// TIA Portal project "Green_Finished" (V17)
// Vorlageprojekt für das Buch mit Zielsystem S7-1200

(* hardware
DEVICE "S7-1200-Station_1"  S7-1200 Station
   slot 0: "Baugruppenträger_0"  Rack  V1.0
   slot 1: "PLC_1"  CPU 1211C DC/DC/DC  6ES7 211-1AE40-0XB0  V4.1
*)

// ===== PLC "PLC_1"  CPU 1211C DC/DC/DC =====

VAR_GLOBAL   // PLC tag table "Standard-Variablentabelle"
   "Tag_1" AT %M0.0 : Bool;
   "Tag_2" AT %M0.1 : Bool;
   "Tag_3" AT %M0.2 : Bool;
   "Tag_4" AT %M0.3 : Bool;
   "Tag_5" AT %M0.4 : Bool;
   "Tag_6" AT %M0.5 : Bool;
   "Tag_7" AT %M0.6 : Bool;
   "vision 0" AT %I2.2 : Bool;
   "arm 0 turn" AT %Q1.5 : Bool;
   "arm 0 +" AT %Q1.6 : Bool;
   "arm 1 turn" AT %Q1.7 : Bool;
   "arm 1 +" AT %Q2.0 : Bool;
   "arm 2 turn" AT %Q2.1 : Bool;
   "arm 2 +" AT %Q2.2 : Bool;
   "6m belt 1" AT %Q2.3 : Bool;
   "curved belt 1" AT %Q2.4 : Bool;
   "4m belt 2" AT %Q2.6 : Bool;
   "vision difuse" AT %I2.3 : Bool;
   "machine 0 produce lid" AT %Q3.1 : Bool;
   "machine 0 start" AT %Q3.2 : Bool;
   "macine 0 stop" AT %Q3.3 : Bool;
   "machine busy" AT %I1.7 : Bool;
   "machine 1 start" AT %Q3.5 : Bool;
   "machine 1 stop" AT %Q3.6 : Bool;
   "machine 1 produce lid" AT %Q3.4 : Bool;
   "curved belt 3" AT %Q4.2 : Bool;
   "curved belt 2" AT %Q4.1 : Bool;
   "6m belt 3" AT %Q4.0 : Bool;
   "6m belt 2" AT %Q3.7 : Bool;
   "4m belt 3" AT %Q3.0 : Bool;
   "2m belt 1" AT %Q2.7 : Bool;
   "2m belt 0" AT %Q2.5 : Bool;
   "diffuse belt 1" AT %I1.6 : Bool;
   "diffuse belt 1 second" AT %I2.5 : Bool;
   "diffuse belt 2" AT %I2.1 : Bool;
   "diffuse belt 2 second" AT %I2.4 : Bool;
   "machine 2 produce lid" AT %Q4.3 : Bool;
   "machine 2 start" AT %Q4.4 : Bool;
   "machine 2 stop" AT %Q4.5 : Bool;
   "machine 3 produce lid" AT %Q4.6 : Bool;
   "machine 3 start" AT %Q4.7 : Bool;
   "machine 3 stop" AT %Q5.0 : Bool;
   "Tag_8" AT %M3.2 : Bool;
   "Tag_9" AT %M3.3 : Bool;
   "Tag_10" AT %M8.0 : Bool;
   "Tag_11" AT %M3.4 : Bool;
   "Tag_12" AT %M3.5 : Bool;
   "Tag_13" AT %M3.6 : Bool;
   "Tag_14" AT %M3.7 : Bool;
   "Tag_15" AT %M4.0 : Bool;
END_VAR

VAR_GLOBAL   // PLC tag table "Sensors & Pushbuttons"
   "Start" AT %I0.0 : Bool;
   "Stop" AT %I0.1 : Bool;
   "Emergency Stop" AT %I0.2 : Bool;
   "RobotDetect" AT %I0.3 : Bool;
   "Diffuser 1" AT %I0.4 : Bool;
   "Diffuser 2" AT %I0.5 : Bool;
   "Frontlimit0" AT %I0.6 : Bool;
   "Backlimit0" AT %I0.7 : Bool;
   "Frontlimit1" AT %I1.0 : Bool;
   "Backlimit1" AT %I1.1 : Bool;
   "Diffuser 3" AT %I1.2 : Bool;
   "Zmoving" AT %I1.3 : Bool;
   "Xmoving" AT %I1.4 : Bool;
   "OBJheld" AT %I1.5 : Bool;
   "Diffuser 9" AT %I3.0 : Bool;
   "Diffuser 10" AT %I3.1 : Bool;
   "Diffuser 13" AT %I3.2 : Bool;
   "Diffuser 14" AT %I3.3 : Bool;
   "Robot1zmoving" AT %I3.4 : Bool;
   "Robot1Xmoving" AT %I3.5 : Bool;
   "ClamperLimit" AT %I4.0 : Bool;
   "ClamperClamped" AT %I4.1 : Bool;
   "Robot1Detected" AT %I3.6 : Bool;
   "Diffuser 17" AT %I4.2 : Bool;
   "Diiffuser 18" AT %I4.3 : Bool;
END_VAR

VAR_GLOBAL   // PLC tag table "Actuators"
   "FeedingConveyer" AT %Q0.0 : Bool;
   "Bridge" AT %Q0.1 : Bool;
   "To machine" AT %Q0.2 : Bool;
   "CurvedConveyer" AT %Q0.3 : Bool;
   "Emitter" AT %Q0.4 : Bool;
   "Pusher0" AT %Q0.5 : Bool;
   "Pusher1" AT %Q0.6 : Bool;
   "GreenLight" AT %Q0.7 : Bool;
   "RedLight" AT %Q1.0 : Bool;
   "Xcontrol" AT %Q1.1 : Bool;
   "Zcontrol" AT %Q1.2 : Bool;
   "Grab" AT %Q1.3 : Bool;
   "WarningLight" AT %Q1.4 : Bool;
   "Belt4m4" AT %Q5.5 : Bool;
   "Belt4m8" AT %Q5.6 : Bool;
   "Cbc4cw" AT %Q5.7 : Bool;
   "Belt6m4" AT %Q6.0 : Bool;
   "Belt4m5" AT %Q6.2 : Bool;
   "CBC5cw" AT %Q6.3 : Bool;
   "Belt2m2" AT %Q6.4 : Bool;
   "cbc5ccw" AT %Q6.5 : Bool;
   "belt6m5" AT %Q6.6 : Bool;
   "Robot1z" AT %Q7.0 : Bool;
   "Robot1x" AT %Q7.5 : Bool;
   "Robot1grab" AT %Q7.3 : Bool;
   "ClamperRaise" AT %Q8.1 : Bool;
   "ClamperClamp" AT %Q8.0 : Bool;
END_VAR

FUNCTION "MHJ-PLC-Lab-Function-S71200" : Void   // FC9000, SCL
{ S7_Optimized_Access := 'TRUE' }
VERSION : 0.1
   VAR_TEMP
      rdTimeReturn : Int;
      outputTime : DTL;
      SyncVal : Byte;
      forVal : Int;
      forVal_2 : Int;
      Value : Byte;
   END_VAR
   VAR CONSTANT
      CompVal : Byte := 16#34;
      Value_01 : Byte := 16#11;
      Value_01_DW : DWord := 16#A165_D992;
      Value_02_DW : DWord := 16#58BE_4401;
   END_VAR
BEGIN

   #Value:=PEEK(area := 16#82,
        dbNumber := 0,
        byteOffset := 511);
   #Value := #Value + 1;

   POKE(area := 16#82,
        dbNumber := 0,
        byteOffset := 511,
        value := #Value);

   POKE(area:=16#81,
        dbNumber:=0,
        byteOffset:=1016,
        value:=#Value_01_DW);
   POKE(area := 16#81,
        dbNumber := 0,
        byteOffset := 1020,
        value := #Value_02_DW);

   POKE(area := 16#81,
        dbNumber := 0,
        byteOffset := 511,
        value := B#16#00);

   FOR #forVal := 0 TO 120 DO
       FOR #forVal_2:=0 TO 10 DO
           #rdTimeReturn:=RD_SYS_T(#outputTime);
           #rdTimeReturn := WR_SYS_T(#outputTime);
           #rdTimeReturn := RD_SYS_T(#outputTime);
           #rdTimeReturn := WR_SYS_T(#outputTime);
       END_FOR;
       #SyncVal:= PEEK(area := 16#81,
                      dbNumber := 0,
                      byteOffset := 511);
       IF #SyncVal = #CompVal THEN
          GOTO M_1;
       END_IF;
   END_FOR;
   RETURN;

   M_1:
   POKE(area := 16#81,
        dbNumber := 0,
        byteOffset := 511,
        value := B#16#0);
END_FUNCTION

ORGANIZATION_BLOCK "Main"   // OB1, LAD, ProgramCycle
TITLE = "Main Program Sweep (Cycle)"
{ S7_Optimized_Access := 'TRUE' }
VERSION : 0.1
   VAR_INPUT
      Initial_Call : Bool;   // Initial call of this OB
      Remanence : Bool;   // =True, if remanent data are available
   END_VAR
   VAR_TEMP   // added for the SCL form of the ladder/FBD networks
      _w1 : Bool;
      _w2 : Bool;
      _w3 : Bool;
      _w4 : Bool;
      _w5 : Bool;
   END_VAR
BEGIN

REGION Network 1: Konnektierungsbaustein für PLC-Lab
   // Im Netzwerk 1 wird der Konnektierungsbaustein für PLC-Lab aufgerufen.
   // Dieser Aufruf darf nicht entfernt werden!
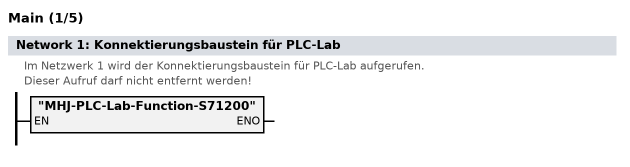
   RUNG wire#powerrail
      "MHJ-PLC-Lab-Function-S71200"()
   END_RUNG
   // the same network as SCL:
   "MHJ-PLC-Lab-Function-S71200"();
END_REGION

REGION Network 2: Ihr Programm / Conveyer Control
   // Schreiben Sie ab Netzwerk 2 Ihr Programm
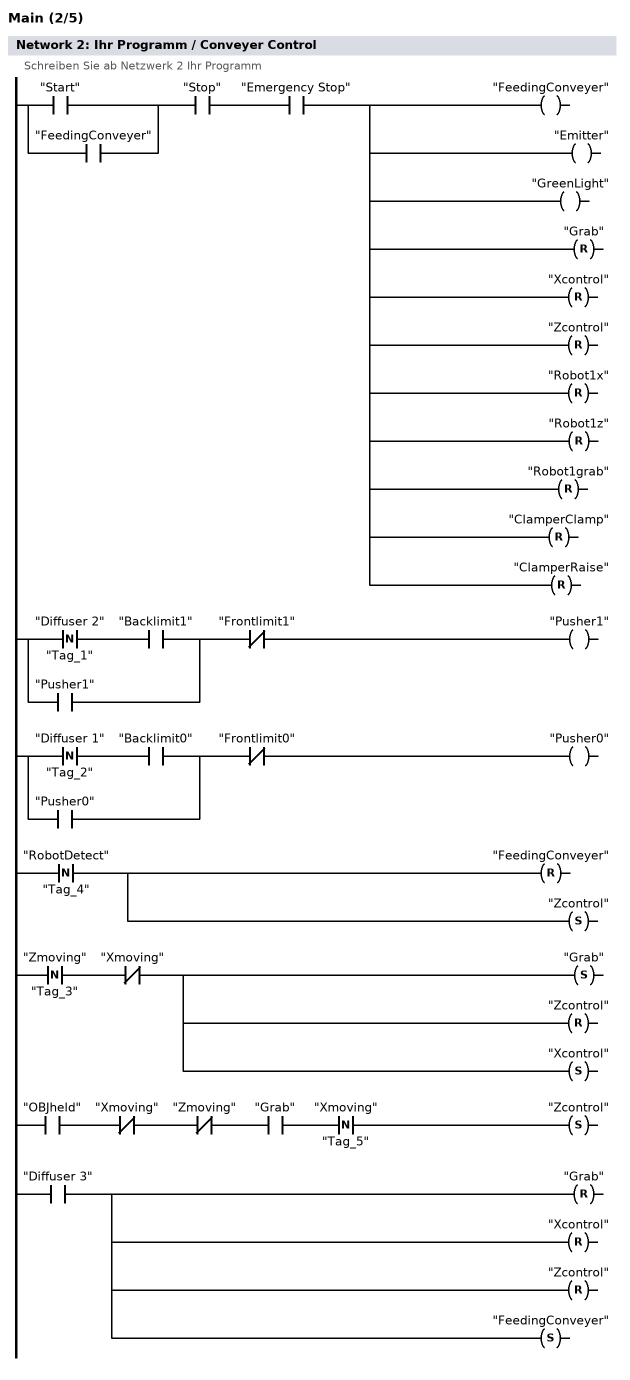
   RUNG wire#powerrail
      Contact( "Start" )
      wire#w1
      Contact( "Stop" )
      Contact( "Emergency Stop" )
      wire#w2
      Coil( "FeedingConveyer" )
   END_RUNG
   RUNG wire#powerrail
      Contact( "FeedingConveyer" )
   END_RUNG wire#w1
   RUNG wire#w2
      Coil( "Emitter" )
   END_RUNG
   RUNG wire#w2
      Coil( "GreenLight" )
   END_RUNG
   RUNG wire#w2
      R_Coil( "Grab" )
   END_RUNG
   RUNG wire#w2
      R_Coil( "Xcontrol" )
   END_RUNG
   RUNG wire#w2
      R_Coil( "Zcontrol" )
   END_RUNG
   RUNG wire#w2
      R_Coil( "Robot1x" )
   END_RUNG
   RUNG wire#w2
      R_Coil( "Robot1z" )
   END_RUNG
   RUNG wire#w2
      R_Coil( "Robot1grab" )
   END_RUNG
   RUNG wire#w2
      R_Coil( "ClamperClamp" )
   END_RUNG
   RUNG wire#w2
      R_Coil( "ClamperRaise" )
   END_RUNG
   RUNG wire#powerrail
      N_Contact(operand := "Diffuser 2", bit := "Tag_1")
      Contact( "Backlimit1" )
      wire#w3
      I_Contact( "Frontlimit1" )
      Coil( "Pusher1" )
   END_RUNG
   RUNG wire#powerrail
      Contact( "Pusher1" )
   END_RUNG wire#w3
   RUNG wire#powerrail
      N_Contact(operand := "Diffuser 1", bit := "Tag_2")
      Contact( "Backlimit0" )
      wire#w4
      I_Contact( "Frontlimit0" )
      Coil( "Pusher0" )
   END_RUNG
   RUNG wire#powerrail
      Contact( "Pusher0" )
   END_RUNG wire#w4
   RUNG wire#powerrail
      N_Contact(operand := "RobotDetect", bit := "Tag_4")
      wire#w5
      R_Coil( "FeedingConveyer" )
   END_RUNG
   RUNG wire#w5
      S_Coil( "Zcontrol" )
   END_RUNG
   RUNG wire#powerrail
      N_Contact(operand := "Zmoving", bit := "Tag_3")
      I_Contact( "Xmoving" )
      wire#w6
      S_Coil( "Grab" )
   END_RUNG
   RUNG wire#w6
      R_Coil( "Zcontrol" )
   END_RUNG
   RUNG wire#w6
      S_Coil( "Xcontrol" )
   END_RUNG
   RUNG wire#powerrail
      Contact( "OBJheld" )
      I_Contact( "Xmoving" )
      I_Contact( "Zmoving" )
      Contact( "Grab" )
      N_Contact(operand := "Xmoving", bit := "Tag_5")
      S_Coil( "Zcontrol" )
   END_RUNG
   RUNG wire#powerrail
      Contact( "Diffuser 3" )
      wire#w7
      R_Coil( "Grab" )
   END_RUNG
   RUNG wire#w7
      R_Coil( "Xcontrol" )
   END_RUNG
   RUNG wire#w7
      R_Coil( "Zcontrol" )
   END_RUNG
   RUNG wire#w7
      S_Coil( "FeedingConveyer" )
   END_RUNG
   // the same network as SCL:
   "FeedingConveyer" := ("Start" OR "FeedingConveyer") AND "Stop" AND "Emergency Stop";
   "Emitter" := "FeedingConveyer";
   "GreenLight" := "FeedingConveyer";
   IF "FeedingConveyer" THEN
       "Grab" := FALSE;
       "Xcontrol" := FALSE;
       "Zcontrol" := FALSE;
       "Robot1x" := FALSE;
       "Robot1z" := FALSE;
       "Robot1grab" := FALSE;
       "ClamperClamp" := FALSE;
       "ClamperRaise" := FALSE;
   END_IF;
   #_w1 := NOT "Diffuser 2" AND "Tag_1";   // falling edge of "Diffuser 2"
   "Tag_1" := "Diffuser 2";
   "Pusher1" := ((#_w1 AND "Backlimit1") OR "Pusher1") AND NOT "Frontlimit1";
   #_w2 := NOT "Diffuser 1" AND "Tag_2";   // falling edge of "Diffuser 1"
   "Tag_2" := "Diffuser 1";
   "Pusher0" := ((#_w2 AND "Backlimit0") OR "Pusher0") AND NOT "Frontlimit0";
   #_w3 := NOT "RobotDetect" AND "Tag_4";   // falling edge of "RobotDetect"
   "Tag_4" := "RobotDetect";
   IF #_w3 THEN
       "FeedingConveyer" := FALSE;
       "Zcontrol" := TRUE;
   END_IF;
   #_w4 := NOT "Zmoving" AND "Tag_3";   // falling edge of "Zmoving"
   "Tag_3" := "Zmoving";
   IF #_w4 AND NOT "Xmoving" THEN
       "Grab" := TRUE;
       "Zcontrol" := FALSE;
       "Xcontrol" := TRUE;
   END_IF;
   #_w5 := "OBJheld" AND NOT "Xmoving" AND NOT "Zmoving" AND "Grab" AND NOT "Xmoving" AND "Tag_5";   // falling edge of "Xmoving"
   "Tag_5" := "Xmoving";
   IF #_w5 THEN "Zcontrol" := TRUE; END_IF;
   IF "Diffuser 3" THEN
       "Grab" := FALSE;
       "Xcontrol" := FALSE;
       "Zcontrol" := FALSE;
       "FeedingConveyer" := TRUE;
   END_IF;
END_REGION

REGION Network 3
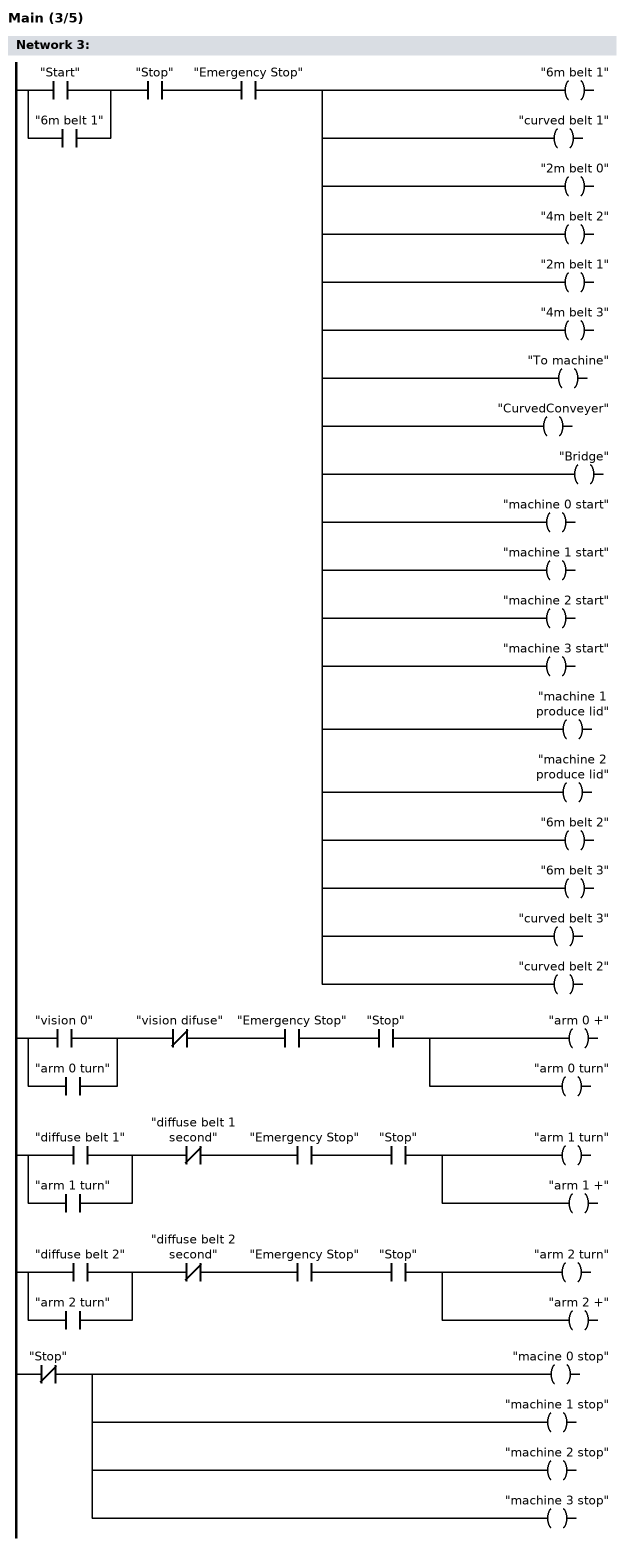
   RUNG wire#powerrail
      Contact( "Start" )
      wire#w1
      Contact( "Stop" )
      Contact( "Emergency Stop" )
      wire#w2
      Coil( "6m belt 1" )
   END_RUNG
   RUNG wire#powerrail
      Contact( "6m belt 1" )
   END_RUNG wire#w1
   RUNG wire#w2
      Coil( "curved belt 1" )
   END_RUNG
   RUNG wire#w2
      Coil( "2m belt 0" )
   END_RUNG
   RUNG wire#w2
      Coil( "4m belt 2" )
   END_RUNG
   RUNG wire#w2
      Coil( "2m belt 1" )
   END_RUNG
   RUNG wire#w2
      Coil( "4m belt 3" )
   END_RUNG
   RUNG wire#w2
      Coil( "To machine" )
   END_RUNG
   RUNG wire#w2
      Coil( "CurvedConveyer" )
   END_RUNG
   RUNG wire#w2
      Coil( "Bridge" )
   END_RUNG
   RUNG wire#w2
      Coil( "machine 0 start" )
   END_RUNG
   RUNG wire#w2
      Coil( "machine 1 start" )
   END_RUNG
   RUNG wire#w2
      Coil( "machine 2 start" )
   END_RUNG
   RUNG wire#w2
      Coil( "machine 3 start" )
   END_RUNG
   RUNG wire#w2
      Coil( "machine 1 produce lid" )
   END_RUNG
   RUNG wire#w2
      Coil( "machine 2 produce lid" )
   END_RUNG
   RUNG wire#w2
      Coil( "6m belt 2" )
   END_RUNG
   RUNG wire#w2
      Coil( "6m belt 3" )
   END_RUNG
   RUNG wire#w2
      Coil( "curved belt 3" )
   END_RUNG
   RUNG wire#w2
      Coil( "curved belt 2" )
   END_RUNG
   RUNG wire#powerrail
      Contact( "vision 0" )
      wire#w3
      I_Contact( "vision difuse" )
      Contact( "Emergency Stop" )
      Contact( "Stop" )
      wire#w4
      Coil( "arm 0 +" )
   END_RUNG
   RUNG wire#powerrail
      Contact( "arm 0 turn" )
   END_RUNG wire#w3
   RUNG wire#w4
      Coil( "arm 0 turn" )
   END_RUNG
   RUNG wire#powerrail
      Contact( "diffuse belt 1" )
      wire#w5
      I_Contact( "diffuse belt 1 second" )
      Contact( "Emergency Stop" )
      Contact( "Stop" )
      wire#w6
      Coil( "arm 1 turn" )
   END_RUNG
   RUNG wire#powerrail
      Contact( "arm 1 turn" )
   END_RUNG wire#w5
   RUNG wire#w6
      Coil( "arm 1 +" )
   END_RUNG
   RUNG wire#powerrail
      Contact( "diffuse belt 2" )
      wire#w7
      I_Contact( "diffuse belt 2 second" )
      Contact( "Emergency Stop" )
      Contact( "Stop" )
      wire#w8
      Coil( "arm 2 turn" )
   END_RUNG
   RUNG wire#powerrail
      Contact( "arm 2 turn" )
   END_RUNG wire#w7
   RUNG wire#w8
      Coil( "arm 2 +" )
   END_RUNG
   RUNG wire#powerrail
      I_Contact( "Stop" )
      wire#w9
      Coil( "macine 0 stop" )
   END_RUNG
   RUNG wire#w9
      Coil( "machine 1 stop" )
   END_RUNG
   RUNG wire#w9
      Coil( "machine 2 stop" )
   END_RUNG
   RUNG wire#w9
      Coil( "machine 3 stop" )
   END_RUNG
   // the same network as SCL:
   "6m belt 1" := ("Start" OR "6m belt 1") AND "Stop" AND "Emergency Stop";
   "curved belt 1" := "6m belt 1";
   "2m belt 0" := "6m belt 1";
   "4m belt 2" := "6m belt 1";
   "2m belt 1" := "6m belt 1";
   "4m belt 3" := "6m belt 1";
   "To machine" := "6m belt 1";
   "CurvedConveyer" := "6m belt 1";
   "Bridge" := "6m belt 1";
   "machine 0 start" := "6m belt 1";
   "machine 1 start" := "6m belt 1";
   "machine 2 start" := "6m belt 1";
   "machine 3 start" := "6m belt 1";
   "machine 1 produce lid" := "6m belt 1";
   "machine 2 produce lid" := "6m belt 1";
   "6m belt 2" := "6m belt 1";
   "6m belt 3" := "6m belt 1";
   "curved belt 3" := "6m belt 1";
   "curved belt 2" := "6m belt 1";
   "arm 0 +" := ("vision 0" OR "arm 0 turn") AND NOT "vision difuse" AND "Emergency Stop" AND "Stop";
   "arm 0 turn" := "arm 0 +";
   "arm 1 turn" := ("diffuse belt 1" OR "arm 1 turn") AND NOT "diffuse belt 1 second" AND "Emergency Stop" AND "Stop";
   "arm 1 +" := "arm 1 turn";
   "arm 2 turn" := ("diffuse belt 2" OR "arm 2 turn") AND NOT "diffuse belt 2 second" AND "Emergency Stop" AND "Stop";
   "arm 2 +" := "arm 2 turn";
   "macine 0 stop" := NOT "Stop";
   "machine 1 stop" := NOT "Stop";
   "machine 2 stop" := NOT "Stop";
   "machine 3 stop" := NOT "Stop";
END_REGION

REGION Network 4
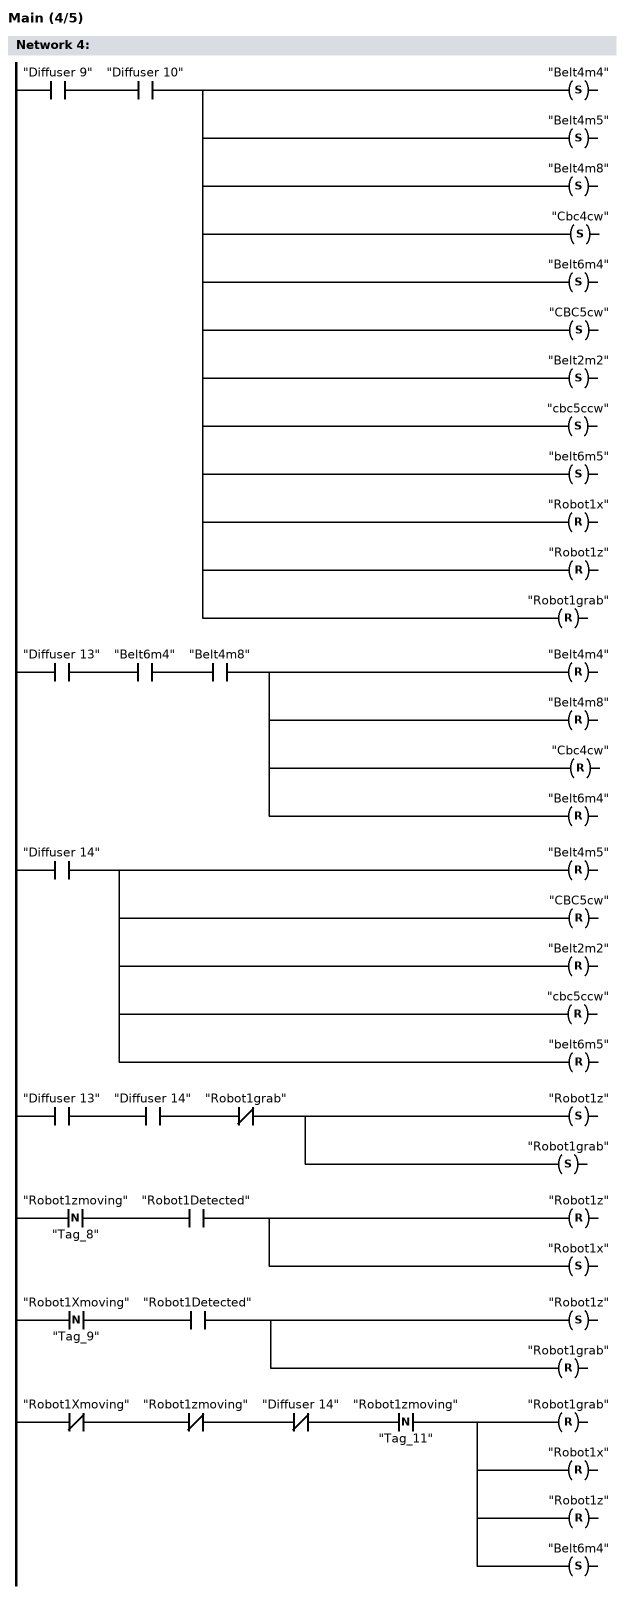
   RUNG wire#powerrail
      Contact( "Diffuser 9" )
      Contact( "Diffuser 10" )
      wire#w1
      S_Coil( "Belt4m4" )
   END_RUNG
   RUNG wire#w1
      S_Coil( "Belt4m5" )
   END_RUNG
   RUNG wire#w1
      S_Coil( "Belt4m8" )
   END_RUNG
   RUNG wire#w1
      S_Coil( "Cbc4cw" )
   END_RUNG
   RUNG wire#w1
      S_Coil( "Belt6m4" )
   END_RUNG
   RUNG wire#w1
      S_Coil( "CBC5cw" )
   END_RUNG
   RUNG wire#w1
      S_Coil( "Belt2m2" )
   END_RUNG
   RUNG wire#w1
      S_Coil( "cbc5ccw" )
   END_RUNG
   RUNG wire#w1
      S_Coil( "belt6m5" )
   END_RUNG
   RUNG wire#w1
      R_Coil( "Robot1x" )
   END_RUNG
   RUNG wire#w1
      R_Coil( "Robot1z" )
   END_RUNG
   RUNG wire#w1
      R_Coil( "Robot1grab" )
   END_RUNG
   RUNG wire#powerrail
      Contact( "Diffuser 13" )
      Contact( "Belt6m4" )
      Contact( "Belt4m8" )
      wire#w2
      R_Coil( "Belt4m4" )
   END_RUNG
   RUNG wire#w2
      R_Coil( "Belt4m8" )
   END_RUNG
   RUNG wire#w2
      R_Coil( "Cbc4cw" )
   END_RUNG
   RUNG wire#w2
      R_Coil( "Belt6m4" )
   END_RUNG
   RUNG wire#powerrail
      Contact( "Diffuser 14" )
      wire#w3
      R_Coil( "Belt4m5" )
   END_RUNG
   RUNG wire#w3
      R_Coil( "CBC5cw" )
   END_RUNG
   RUNG wire#w3
      R_Coil( "Belt2m2" )
   END_RUNG
   RUNG wire#w3
      R_Coil( "cbc5ccw" )
   END_RUNG
   RUNG wire#w3
      R_Coil( "belt6m5" )
   END_RUNG
   RUNG wire#powerrail
      Contact( "Diffuser 13" )
      Contact( "Diffuser 14" )
      I_Contact( "Robot1grab" )
      wire#w4
      S_Coil( "Robot1z" )
   END_RUNG
   RUNG wire#w4
      S_Coil( "Robot1grab" )
   END_RUNG
   RUNG wire#powerrail
      N_Contact(operand := "Robot1zmoving", bit := "Tag_8")
      Contact( "Robot1Detected" )
      wire#w5
      R_Coil( "Robot1z" )
   END_RUNG
   RUNG wire#w5
      S_Coil( "Robot1x" )
   END_RUNG
   RUNG wire#powerrail
      N_Contact(operand := "Robot1Xmoving", bit := "Tag_9")
      Contact( "Robot1Detected" )
      wire#w6
      S_Coil( "Robot1z" )
   END_RUNG
   RUNG wire#w6
      R_Coil( "Robot1grab" )
   END_RUNG
   RUNG wire#powerrail
      I_Contact( "Robot1Xmoving" )
      I_Contact( "Robot1zmoving" )
      I_Contact( "Diffuser 14" )
      N_Contact(operand := "Robot1zmoving", bit := "Tag_11")
      wire#w7
      R_Coil( "Robot1grab" )
   END_RUNG
   RUNG wire#w7
      R_Coil( "Robot1x" )
   END_RUNG
   RUNG wire#w7
      R_Coil( "Robot1z" )
   END_RUNG
   RUNG wire#w7
      S_Coil( "Belt6m4" )
   END_RUNG
   // the same network as SCL:
   IF "Diffuser 9" AND "Diffuser 10" THEN
       "Belt4m4" := TRUE;
       "Belt4m5" := TRUE;
       "Belt4m8" := TRUE;
       "Cbc4cw" := TRUE;
       "Belt6m4" := TRUE;
       "CBC5cw" := TRUE;
       "Belt2m2" := TRUE;
       "cbc5ccw" := TRUE;
       "belt6m5" := TRUE;
       "Robot1x" := FALSE;
       "Robot1z" := FALSE;
       "Robot1grab" := FALSE;
   END_IF;
   IF "Diffuser 13" AND "Belt6m4" AND "Belt4m8" THEN "Belt4m4" := FALSE; END_IF;
   #_w1 := "Diffuser 13" AND "Belt6m4" AND "Belt4m8";
   IF #_w1 THEN
       "Belt4m8" := FALSE;
       "Cbc4cw" := FALSE;
       "Belt6m4" := FALSE;
   END_IF;
   IF "Diffuser 14" THEN
       "Belt4m5" := FALSE;
       "CBC5cw" := FALSE;
       "Belt2m2" := FALSE;
       "cbc5ccw" := FALSE;
       "belt6m5" := FALSE;
   END_IF;
   IF "Diffuser 13" AND "Diffuser 14" AND NOT "Robot1grab" THEN
       "Robot1z" := TRUE;
       "Robot1grab" := TRUE;
   END_IF;
   #_w2 := NOT "Robot1zmoving" AND "Tag_8";   // falling edge of "Robot1zmoving"
   "Tag_8" := "Robot1zmoving";
   IF #_w2 AND "Robot1Detected" THEN
       "Robot1z" := FALSE;
       "Robot1x" := TRUE;
   END_IF;
   #_w3 := NOT "Robot1Xmoving" AND "Tag_9";   // falling edge of "Robot1Xmoving"
   "Tag_9" := "Robot1Xmoving";
   IF #_w3 AND "Robot1Detected" THEN
       "Robot1z" := TRUE;
       "Robot1grab" := FALSE;
   END_IF;
   #_w4 := NOT "Robot1Xmoving" AND NOT "Robot1zmoving" AND NOT "Diffuser 14" AND NOT "Robot1zmoving" AND "Tag_11";   // falling edge of "Robot1zmoving"
   "Tag_11" := "Robot1zmoving";
   IF #_w4 THEN
       "Robot1grab" := FALSE;
       "Robot1x" := FALSE;
       "Robot1z" := FALSE;
       "Belt6m4" := TRUE;
   END_IF;
END_REGION

REGION Network 5
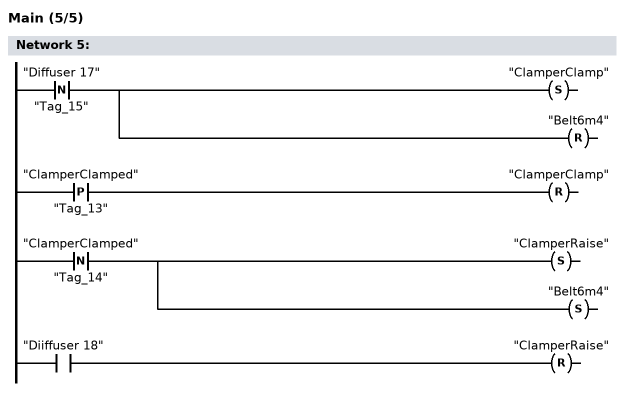
   RUNG wire#powerrail
      N_Contact(operand := "Diffuser 17", bit := "Tag_15")
      wire#w1
      S_Coil( "ClamperClamp" )
   END_RUNG
   RUNG wire#w1
      R_Coil( "Belt6m4" )
   END_RUNG
   RUNG wire#powerrail
      P_Contact(operand := "ClamperClamped", bit := "Tag_13")
      R_Coil( "ClamperClamp" )
   END_RUNG
   RUNG wire#powerrail
      N_Contact(operand := "ClamperClamped", bit := "Tag_14")
      wire#w2
      S_Coil( "ClamperRaise" )
   END_RUNG
   RUNG wire#w2
      S_Coil( "Belt6m4" )
   END_RUNG
   RUNG wire#powerrail
      Contact( "Diiffuser 18" )
      R_Coil( "ClamperRaise" )
   END_RUNG
   // the same network as SCL:
   #_w1 := NOT "Diffuser 17" AND "Tag_15";   // falling edge of "Diffuser 17"
   "Tag_15" := "Diffuser 17";
   IF #_w1 THEN
       "ClamperClamp" := TRUE;
       "Belt6m4" := FALSE;
   END_IF;
   #_w2 := "ClamperClamped" AND NOT "Tag_13";   // rising edge of "ClamperClamped"
   "Tag_13" := "ClamperClamped";
   IF #_w2 THEN "ClamperClamp" := FALSE; END_IF;
   #_w3 := NOT "ClamperClamped" AND "Tag_14";   // falling edge of "ClamperClamped"
   "Tag_14" := "ClamperClamped";
   IF #_w3 THEN
       "ClamperRaise" := TRUE;
       "Belt6m4" := TRUE;
   END_IF;
   IF "Diiffuser 18" THEN "ClamperRaise" := FALSE; END_IF;
END_REGION
END_ORGANIZATION_BLOCK